{attribute addProperty BoxType "EP1816-3008-0016"}
{attribute addProperty Id "DIG_Inputs_ChannelAT %I*ARRAY[0..8] OF DIG_Inputs_Channel_628B507D128160AI_Inputs_ChannelAT %I*ARRAY[0..10] OF AI_Inputs_Channel_36527000192240DIG_Inputs_DeviceAT %I*DIG_Inputs_Device_5061D9393240WcStateAT %I*WcState_98A4DF7520.250InfoDataAT %I*InfoData_BC63D37F80100"}
{attribute addProperty CRC "3767454239"}
{attribute addProperty SizeInBites "434"}
{attribute addProperty SizeInBytes "54.25"}
TYPE EP1816_F6DE3BA6 :
STRUCT
	{attribute addProperty Name "DIG_Inputs_Channel"}
	DIG_Inputs_Channel : ARRAY[0..8] OF DIG_Inputs_Channel_628B507D;
	{attribute addProperty Name "AI_Inputs_Channel"}
	AI_Inputs_Channel : ARRAY[0..10] OF AI_Inputs_Channel_36527000;
	{attribute addProperty Name "DIG_Inputs_Device"}
	DIG_Inputs_Device : DIG_Inputs_Device_5061D939;
	{attribute addProperty Name "WcState"}
	WcState : WcState_98A4DF75;
	{attribute addProperty Name "InfoData"}
	InfoData : InfoData_BC63D37F;
END_STRUCT
END_TYPE

(* stored: Version 1.2.0.0, ProductVersion 3.1.4024.9
   DUT EP1816_F6DE3BA6: Id {5be27c50-fde0-491b-8ca3-ca25677b4c70} *)
